FUNCTION_BLOCK MotorManagement
VAR_IN_OUT
	Motor	: stMotor;
END_VAR

VAR_INPUT
	xIn_StatusDispatch	: BOOL;
	xIn_StatusError		: BOOL;
	xIn_StatusRunning	: BOOL;
	xIn_ResetError		: BOOL;
	xIn_AuxPower		: BOOL;
	UseReverse			: BOOL;
	TestMode			: BOOL;
	TriggerForward		: BOOL;
	TriggerReverse		: BOOL;
	
END_VAR
VAR_OUTPUT
	Error	: BOOL;
	ErrorID	: UINT;
END_VAR
VAR PERSISTENT
	StatusError			: BOOL;
	MotorCannotRunning	: BOOL;
	PowerOff			: BOOL;
	Timer				: TON;
	LocalSwitch_Off		: BOOL;
	SeqCal				: INT;
	tRunningHours		: LTIME;
	RunningTimer		: LTON;
	lrealRunningHours	: LREAL;
END_VAR
VAR // added by the converter: edge detectors and wires of the graphical bodies
    _w1 : BOOL;
END_VAR

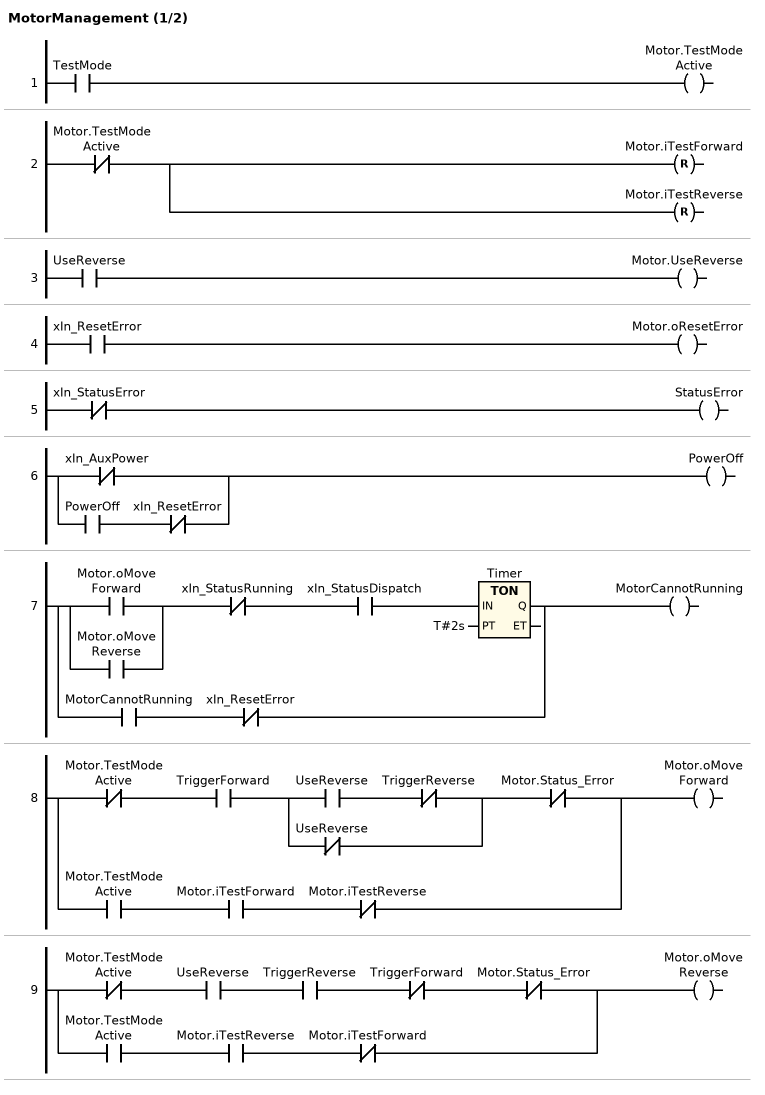
// NETWORK 1
Motor.TestModeActive := TestMode;

// NETWORK 2
_w1 := NOT Motor.TestModeActive;
Motor.iTestForward R= _w1;
Motor.iTestReverse R= _w1;

// NETWORK 3
Motor.UseReverse := UseReverse;

// NETWORK 4
Motor.oResetError := xIn_ResetError;

// NETWORK 5
StatusError := NOT xIn_StatusError;

// NETWORK 6
PowerOff := NOT xIn_AuxPower OR PowerOff AND NOT xIn_ResetError;

// NETWORK 7
Timer(IN := (Motor.oMoveForward OR Motor.oMoveReverse) AND NOT xIn_StatusRunning AND xIn_StatusDispatch, PT := T#2s); // TON
MotorCannotRunning := Timer.Q OR MotorCannotRunning AND NOT xIn_ResetError;

// NETWORK 8
Motor.oMoveForward := NOT Motor.TestModeActive AND TriggerForward AND (UseReverse AND NOT TriggerReverse OR NOT UseReverse) AND NOT Motor.Status_Error OR Motor.TestModeActive AND Motor.iTestForward AND NOT Motor.iTestReverse;

// NETWORK 9
Motor.oMoveReverse := NOT Motor.TestModeActive AND UseReverse AND TriggerReverse AND NOT TriggerForward AND NOT Motor.Status_Error OR Motor.TestModeActive AND Motor.iTestReverse AND NOT Motor.iTestForward;

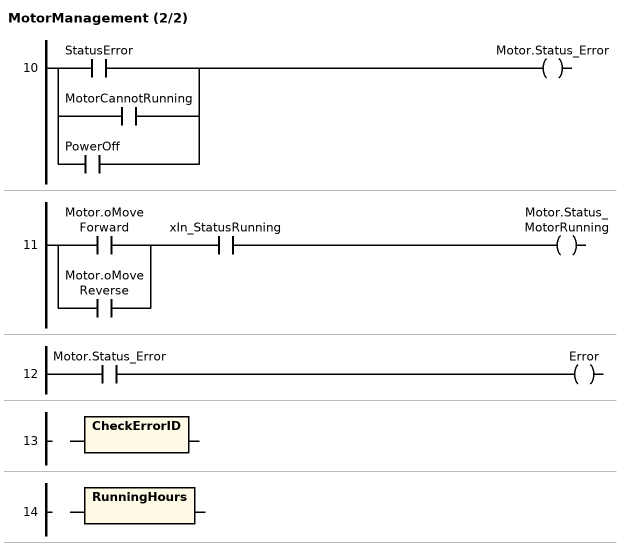
// NETWORK 10
Motor.Status_Error := StatusError OR MotorCannotRunning OR PowerOff;

// NETWORK 11
Motor.Status_MotorRunning := (Motor.oMoveForward OR Motor.oMoveReverse) AND xIn_StatusRunning;

// NETWORK 12
Error := Motor.Status_Error;

// NETWORK 13
CheckErrorID();

// NETWORK 14
RunningHours();

ACTION CheckErrorID:
// Mengatur ErrorID berdasarkan kondisi Error
IF Error THEN
	// Jika ada Error
	IF StatusError THEN
		// Jika StatusError aktif, mengatur ErrorID menjadi 1
		ErrorID:=1;
	ELSIF PowerOff THEN
		// Jika PowerOff aktif, mengatur ErrorID menjadi 2
		ErrorID:=2;
	ELSIF LocalSwitch_Off THEN
		// Jika LocalSwitch_Off aktif, mengatur ErrorID menjadi 3
		ErrorID:=3;
	ELSIF MotorCannotRunning THEN
		// Jika MotorCannotRunning aktif, mengatur ErrorID menjadi 10
		ErrorID:=10;
	ELSE
		// Jika tidak ada kondisi Error yang memenuhi, mengatur ErrorID menjadi 90
		ErrorID:=90;
	END_IF
ELSE
	// Jika tidak ada Error, mengatur ErrorID menjadi 0
	ErrorID:=0;
END_IF

// Mengassign ErrorID ke Motor.ErrorID
Motor.ErrorID:=ErrorID;
END_ACTION

ACTION RunningHours:
// Memilih langkah berdasarkan SeqCal
CASE SeqCal OF
	0:
		// Langkah 0: Mengatur Motor.RunningTime dengan tRunningHours
		Motor.RunningTime := tRunningHours;
		// Jika Status_MotorRunning aktif, lanjut ke langkah 1
		IF Motor.Status_MotorRunning THEN
			SeqCal := 1;
		END_IF
		
	1:
		// Langkah 1: Menghitung waktu berjalan menggunakan RunningTimer
		RunningTimer(IN:=TRUE, PT:=LTIME#1H);
		Motor.RunningTime := tRunningHours + RunningTimer.ET;
		// Jika RunningTimer telah mencapai waktu yang ditetapkan atau Status_MotorRunning tidak aktif, lanjut ke langkah 2
		IF RunningTimer.Q OR NOT Motor.Status_MotorRunning THEN
			RunningTimer(IN:=FALSE);
			SeqCal := 2;
		END_IF
		
	2:
		// Langkah 2: Memperbarui tRunningHours dengan nilai terbaru dari Motor.RunningTime
		tRunningHours := Motor.RunningTime;
		// Kembali ke langkah awal
		SeqCal := 0;
END_CASE

// Mengkonversi Motor.RunningTime ke jam dan menyimpannya di Motor.RunningHours
Motor.RunningHours := LTIME_TO_LREAL(Motor.RunningTime) / LTIME_TO_LREAL(LTIME#1H);
END_ACTION

END_FUNCTION_BLOCK

(* stored: Version 1.1.0.1, ProductVersion 3.1.4024.6
   POU MotorManagement: Id {98de7ba3-21d2-47ac-a773-f5065995e3fd}, SpecialFunc None
   Action CheckErrorID: Id {5f9c736a-4588-46b8-895d-2ff440181742}
   Action RunningHours: Id {fae03b09-f2db-4f7e-9e84-4d4fd28f0412} *)
